FUNCTION_BLOCK FB_Motion
VAR_INPUT

	
END_VAR
VAR_OUTPUT
	
END_VAR
VAR
	fbMcPower	: MC_Power;
	fbMcJog: MC_Jog;
	fbMcMoveAbs: MC_MoveAbsolute;
	fbMcStop: MC_Stop;
	fbMcReset: MC_Reset;
END_VAR

VAR_IN_OUT
	Axis			: AXIS_REF;
	stAxisInterface	: ST_AxisInterface;
	
END_VAR

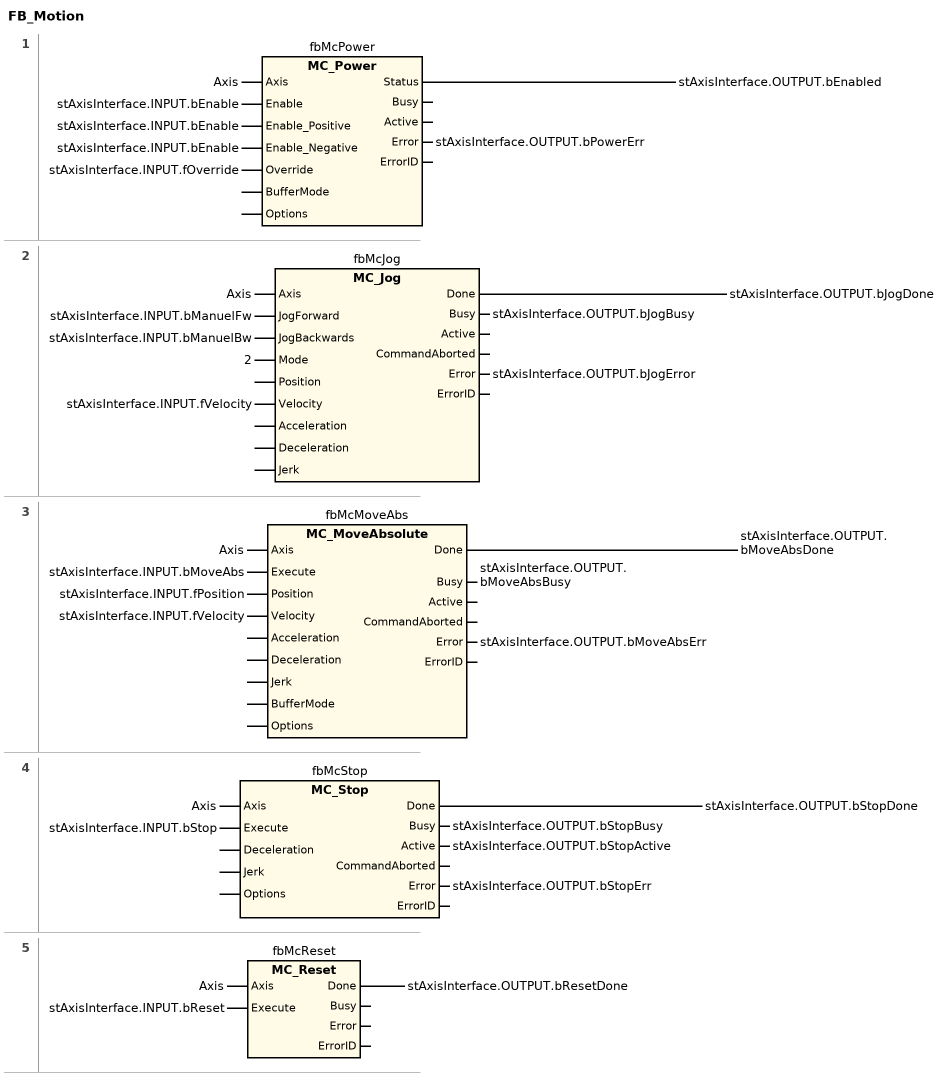
// NETWORK 1
fbMcPower(
    Axis := Axis,
    Enable := stAxisInterface.INPUT.bEnable,
    Enable_Positive := stAxisInterface.INPUT.bEnable,
    Enable_Negative := stAxisInterface.INPUT.bEnable,
    Override := stAxisInterface.INPUT.fOverride,
    Error => stAxisInterface.OUTPUT.bPowerErr); // MC_Power
stAxisInterface.OUTPUT.bEnabled := fbMcPower.Status;

// NETWORK 2
fbMcJog(
    Axis := Axis,
    JogForward := stAxisInterface.INPUT.bManuelFw,
    JogBackwards := stAxisInterface.INPUT.bManuelBw,
    Mode := 2,
    Velocity := stAxisInterface.INPUT.fVelocity,
    Busy => stAxisInterface.OUTPUT.bJogBusy,
    Error => stAxisInterface.OUTPUT.bJogError); // MC_Jog
stAxisInterface.OUTPUT.bJogDone := fbMcJog.Done;

// NETWORK 3
fbMcMoveAbs(
    Axis := Axis,
    Execute := stAxisInterface.INPUT.bMoveAbs,
    Position := stAxisInterface.INPUT.fPosition,
    Velocity := stAxisInterface.INPUT.fVelocity,
    Busy => stAxisInterface.OUTPUT.bMoveAbsBusy,
    Error => stAxisInterface.OUTPUT.bMoveAbsErr); // MC_MoveAbsolute
stAxisInterface.OUTPUT.bMoveAbsDone := fbMcMoveAbs.Done;

// NETWORK 4
fbMcStop(
    Axis := Axis,
    Execute := stAxisInterface.INPUT.bStop,
    Busy => stAxisInterface.OUTPUT.bStopBusy,
    Active => stAxisInterface.OUTPUT.bStopActive,
    Error => stAxisInterface.OUTPUT.bStopErr); // MC_Stop
stAxisInterface.OUTPUT.bStopDone := fbMcStop.Done;

// NETWORK 5
fbMcReset(Axis := Axis, Execute := stAxisInterface.INPUT.bReset); // MC_Reset
stAxisInterface.OUTPUT.bResetDone := fbMcReset.Done;

END_FUNCTION_BLOCK

(* stored: Version 1.1.0.1, ProductVersion 3.1.4022.18
   POU FB_Motion: Id {5a16f141-3300-4b6a-b5ec-6f6450a3cdbe}, SpecialFunc None *)
